PROGRAM main
  VAR
    HS101_STOP : BOOL;
    HS102_START : BOOL;
    M101 : BOOL;
  END_VAR

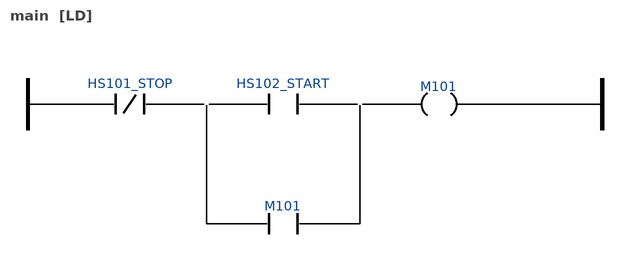
(* LD diagram, written out as Structured Text *)
M101 := NOT HS101_STOP AND (HS102_START OR M101);
END_PROGRAM
